(* IEC 61131-3 sources: JaccoSigma/tempclass/Class/ConnReWr, 1 file *)

(* ---- ConnReWr.st ---- *)
#ifndef cMaxAsciiLine
	#define	cMaxAsciiLine	15 // 1024 //4096	// Max length of an ASCII line
	#define cSeparator		';'			// Separator between two elements
	#define cTestChar		'~'			// Test character
#endif

(*!
<Class
	Name               = "ConnReWr"
	Revision           = "0.0"
	RealtimeTask       = "false"
	CyclicTask         = "true"
	DefCyclictime      = "10 ms"
	BackgroundTask     = "false"
	Sigmatek           = "false"
	OSInterface        = "false"
	HighPriority       = "false"
	Automatic          = "false"
	UpdateMode         = "Prescan"
	SharedCommandTable = "true"
	Objectsize         = "(284,120)">
	<Channels>
		<Server Name="FromNr" Visualized="false" Initialize="false" WriteProtected="false" Retentive="false"/>
		<Server Name="ReadNr" Visualized="false" Initialize="false" WriteProtected="false" Retentive="false"/>
		<Server Name="State" Visualized="false" Initialize="false" WriteProtected="true" Retentive="false"/>
		<Server Name="ToNr" Visualized="false" Initialize="false" WriteProtected="false" Retentive="false"/>
		<Server Name="Value" Visualized="false" Initialize="false" WriteProtected="true" Retentive="false"/>
		<Client Name="In" Required="false" Internal="false"/>
		<Client Name="Out" Required="false" Internal="false"/>
	</Channels>
</Class>
*)
ConnReWr : CLASS
  //Servers:
	Value 	: SvrChCmd_DINT;
	FromNr 	: SvrCh_DINT;
	ToNr 	: SvrCh_DINT;
	ReadNr 	: SvrCh_DINT;
	State 	: SvrCh_DINT;
  //Clients:
	In 	: CltCh_DINT;
	Out 	: CltCh_DINT;
  //Variables:
		RetCode 	: DINT;
		FromName : ARRAY [0..cMaxAsciiLine] OF CHAR;

		ToName : ARRAY [0..cMaxAsciiLine] OF CHAR;

		ReadName : ARRAY [0..cMaxAsciiLine] OF CHAR;

  //Functions:

	FUNCTION VIRTUAL GLOBAL Init;

	FUNCTION VIRTUAL GLOBAL CyWork
		VAR_INPUT
			EAX 	: UDINT;
		END_VAR
		VAR_OUTPUT
			state (EAX) 	: UDINT;
		END_VAR;

	FUNCTION VIRTUAL Connect;

	FUNCTION VIRTUAL BuildFromName;

	FUNCTION VIRTUAL BuildToName;

	FUNCTION VIRTUAL BuildReadName;

	FUNCTION VIRTUAL GLOBAL Value::Read
		VAR_OUTPUT
			output (EAX) 	: DINT;
		END_VAR;

	FUNCTION VIRTUAL GLOBAL FromNr::Write
		VAR_INPUT
			input (EAX) 	: DINT;
		END_VAR
		VAR_OUTPUT
			result (EAX) 	: DINT;
		END_VAR;

	FUNCTION VIRTUAL GLOBAL ToNr::Write
		VAR_INPUT
			input (EAX) 	: DINT;
		END_VAR
		VAR_OUTPUT
			result (EAX) 	: DINT;
		END_VAR;

	FUNCTION VIRTUAL GLOBAL ReadNr::Write
		VAR_INPUT
			input (EAX) 	: DINT;
		END_VAR
		VAR_OUTPUT
			result (EAX) 	: DINT;
		END_VAR;
  //Tables:
	FUNCTION @STD
		VAR_OUTPUT
			ret_code	: CONFSTATES;
		END_VAR;
	FUNCTION GLOBAL TAB @CT_;
END_CLASS;

(*
 * state
 *         0  => OK
 *        -1  => Invalid FromNr
 *        -2  => Invalid ToNr
 *        -3  => Invalid ReadNr
 *        -4  => Invalid return from "ConnectCltSvr()" on server side
 *        -5  => Invalid return from "ConnectCltSvr()" with from name.
 *        -6  => Invalid return from "ConnectCltSvr()" with to name.
 *
 *)

FUNCTION VIRTUAL GLOBAL ConnReWr::Init

  If _FirstScan Then
    FromNr  := 1;
    ToNr    := 1;
    ReadNr  := 1;
    Connect();
  End_If;

END_FUNCTION

FUNCTION VIRTUAL GLOBAL ConnReWr::CyWork
	VAR_INPUT
		EAX 	: UDINT;
	END_VAR
	VAR_OUTPUT
		state (EAX) 	: UDINT;
	END_VAR

  In  := In.Read();
  Out := In;
  Out.Write (Out);

	state := READY;

END_FUNCTION

FUNCTION VIRTUAL GLOBAL ConnReWr::FromNr::Write
	VAR_INPUT
		input (EAX) 	: DINT;
	END_VAR
	VAR_OUTPUT
		result (EAX) 	: DINT;
	END_VAR

	FromNr := input;
  Connect();
 	result := FromNr;

END_FUNCTION

FUNCTION VIRTUAL GLOBAL ConnReWr::ToNr::Write
	VAR_INPUT
		input (EAX) 	: DINT;
	END_VAR
	VAR_OUTPUT
		result (EAX) 	: DINT;
	END_VAR

	ToNr := input;
  Connect();
 	result := ToNr;

END_FUNCTION

FUNCTION VIRTUAL GLOBAL ConnReWr::ReadNr::Write
	VAR_INPUT
		input (EAX) 	: DINT;
	END_VAR
	VAR_OUTPUT
		result (EAX) 	: DINT;
	END_VAR

	ReadNr := input;
  Connect();
 	result := ReadNr;

END_FUNCTION

FUNCTION VIRTUAL ConnReWr::Connect

  state  := 0;
  BuildReadName();
  BuildFromName();
  BuildToName();
  RetCode := ConnectCltSvr( pCltName := #ReadName[0], pSvrName := "ConnReWr.Value");
  if RetCode<> 0 then
    state  := -4;
  else
//    RetCode := ConnectCltSvr( pCltName := "ConnReWr.In1", pSvrName := "In3.Value");
//    RetCode := ConnectCltSvr( pCltName := "ConnReWr.In1", pSvrName := #FromName[0]);
    RetCode := ConnectCltSvr( pCltName := "ConnReWr.In", pSvrName := #FromName[0]);
    if RetCode<> 0 then
      state  := -5;
    else
      RetCode := ConnectCltSvr( pCltName := "ConnReWr.Out", pSvrName := #ToName[0]);
      if RetCode<> 0 then
        state  := -6;
      end_if;
    end_if;
  end_if;

END_FUNCTION

FUNCTION VIRTUAL ConnReWr::BuildFromName

  case FromNr of
  1:
    _MemCpy( #FromName[0], "In1.Value", 10);
  2:
    _MemCpy( #FromName[0], "In2.Value", 10);
  3:  // Test error
    _MemCpy( #FromName[0], "In3.Value", 10);
  else
    state  := -1;
  end_case;

END_FUNCTION

FUNCTION VIRTUAL ConnReWr::BuildToName

  case ToNr of
  1:
    _MemCpy( #ToName[0], "Out1.Data", 10);
  2:
    _MemCpy( #ToName[0], "Out2.Data", 10);
  3:  // Test error
    _MemCpy( #ToName[0], "Out3.Data", 10);
  else
    state  := -2;
  end_case;

END_FUNCTION

FUNCTION VIRTUAL ConnReWr::BuildReadName

  case ReadNr of
  1:
    _MemCpy( #ReadName[0], "Read1.Client_Read", 18);
  2:
    _MemCpy( #ReadName[0], "Read2.Client_Read", 18);
  3:  // Test error
    _MemCpy( #ReadName[0], "Read3.Client_Read", 18);
  else
    state  := -3;
  end_case;

END_FUNCTION

FUNCTION VIRTUAL GLOBAL ConnReWr::Value::Read
	VAR_OUTPUT
		output (EAX) 	: DINT;
	END_VAR

	output := Value := In;

END_FUNCTION
